INTERFACE I_Message

METHOD Send : HRESULT
VAR_INPUT
	Message : T_MaxString;
END_VAR
END_METHOD

END_INTERFACE

(* stored: Version 1.1.0.1
   Itf I_Message: Id {2099f939-9ec3-4558-8ed7-fb5fbee10ec9}
   Method Send: Id {98f2b7ce-6e57-4fac-ac6c-a2745891cfea} *)
